FUNCTION_BLOCK FB_ResetNC_TestDouble IMPLEMENTS  I_Reset
VAR
	bError : BOOL;
	nErrorID : UDINT := 20000;
END_VAR

{warning 'Add property implementation'}
PROPERTY Aborted : BOOL
GET
END_GET
END_PROPERTY

{warning 'Add property implementation'}
PROPERTY Active : BOOL
GET
Active := TRUE;
END_GET
END_PROPERTY

{warning 'Add property implementation'}
PROPERTY Busy : BOOL
GET
END_GET
END_PROPERTY

{warning 'Add property implementation'}
PROPERTY Done : BOOL
GET
END_GET
END_PROPERTY

{warning 'Add property implementation'}
PROPERTY Error : BOOL
GET
Error := bError;
END_GET
SET
bError := Error;
END_SET
END_PROPERTY

{warning 'Add property implementation'}
PROPERTY ErrorID : UDINT
GET
ErrorId := nErrorID;
END_GET
SET
nErrorId := ErrorID;
END_SET
END_PROPERTY

{warning 'Add property implementation'}
PROPERTY Message : T_MAXSTRING
GET
END_GET
END_PROPERTY

{warning 'Add method implementation '}
METHOD Reset
END_METHOD

END_FUNCTION_BLOCK

(* stored: Version 1.1.0.1
   POU FB_ResetNC_TestDouble: Id {4bec94c2-1fc0-49b9-ba47-4c9ac8090ac3}, SpecialFunc None
   Property Aborted: Id {c44d03a4-d22e-42fe-8e82-58b393ba6d2f}
   Get Get: Id {118471bb-28b7-41bc-9627-26a38f6d9399}
   Property Active: Id {5fa2a6b8-e24e-44ea-9d55-fffb9820ab01}
   Get Get: Id {ce24c1d7-df8e-4fd0-8c1c-a9afb9182132}
   Property Busy: Id {61334d3c-93dc-409f-bfb3-3ed8bc09e718}
   Get Get: Id {4b9c2a6b-afeb-4d0b-bb79-b9854f1f2913}
   Property Done: Id {ceadc5dc-060c-488d-bae7-f157c6810b13}
   Get Get: Id {9a1d1d16-8bf6-40e9-85c6-03942c899ee3}
   Property Error: Id {f938065f-d803-4527-8a7e-2dc1fc85c1a0}
   Get Get: Id {ae32733c-1715-491d-a6e4-4ac5b4e14aec}
   Set Set: Id {c8450511-ab84-410d-b1ef-070e191692d8}
   Property ErrorID: Id {d6eac62a-3a87-4a2a-a106-c130598846ef}
   Get Get: Id {645fa3d5-92b4-4e15-908a-70447a9daf13}
   Set Set: Id {bf681c9e-6414-45f2-8d90-9c511a5151dc}
   Property Message: Id {837bcae6-b221-4858-8b6c-574209efce91}
   Get Get: Id {d8cc70db-c18f-4b1b-97bd-30910696c78e}
   Method Reset: Id {baceac4e-8cd9-4713-bb46-b638d35d7dae} *)
